(* CoDeSys 2.3.9.41 project: FirstProg.pro *)
(* Libraries: STANDARD.LIB 5.6.98 12:03:02 *)

(* Task configuration *)
TASK Standard (PRIORITY := 0, INTERVAL := T#5ms);
	MAIN
END_TASK

(* Global variable list: Globale_Variablen *)
	VAR_GLOBAL
	globButtonYellow AT %I* : BOOL;
	globButtonBlue AT %I* : BOOL ;
	globLightGreen AT %Q* : BOOL;
	globLightRed AT %Q*  : BOOL;
	globAnalogOutput AT%Q* : INT;
END_VAR

VAR_GLOBAL
	analogOutputMaxVolt : INT :=10 ;
	intMaxValue : INT := 16#7FFF;
	samplingTime : REAL :=0.005;
END_VAR

(* Global variable list: TwinCAT_Configuration *)
(* Generated automatically by TwinCAT - (read only) *)
VAR_CONFIG
	.globButtonYellow AT %IX0.0 : BOOL;	(*  ~ {LinkedWith:TIID^Device 1 (EtherCAT)^Term 1 (EK1200)^Term 2 (EL1004)^Channel 1^Input} *)
	.globButtonBlue AT %IX0.1 : BOOL;	(*  ~ {LinkedWith:TIID^Device 1 (EtherCAT)^Term 1 (EK1200)^Term 2 (EL1004)^Channel 2^Input} *)
	.globLightGreen AT %QX0.0 : BOOL;	(*  ~ {LinkedWith:TIID^Device 1 (EtherCAT)^Term 1 (EK1200)^Term 3 (EL2004)^Channel 1^Output} *)
	.globLightRed AT %QX0.1 : BOOL;	(*  ~ {LinkedWith:TIID^Device 1 (EtherCAT)^Term 1 (EK1200)^Term 3 (EL2004)^Channel 2^Output} *)
	.globAnalogOutput AT %QB4 : INT;	(*  ~ {LinkedWith:TIID^Device 1 (EtherCAT)^Term 1 (EK1200)^Term 5 (EL4034)^AO Outputs Channel 1^Analog output} *)
END_VAR

(* POU MAIN, ST *)
PROGRAM MAIN
VAR
	myBlock : addBlock;
	test : REAL;
END_VAR
UnserProgramm();
myBlock(a := 6.0, b := 6.0);
END_PROGRAM

(* POU addBlock, ST *)
FUNCTION_BLOCK addBlock
VAR_INPUT
	a : REAL;
	b : REAL;
END_VAR
VAR_OUTPUT
	addition : REAL;
	subtraction : REAL;
END_VAR
VAR
END_VAR
addition := a+b;
subtraction := a-b;
END_FUNCTION_BLOCK

(* POU UnserProgramm, ST *)
PROGRAM UnserProgramm
VAR
	intButtonYellowCount : INT := 0;
	Volt : INT;
END_VAR
IF globButtonYellow = TRUE THEN
	globLightGreen := TRUE;
	intButtonYellowCount := intButtonYellowCount + 1;
ELSE
	globLightGreen := FALSE;
END_IF

IF globButtonBlue = TRUE THEN
	globLightRed := TRUE;
	intButtonYellowCount := 0;
ELSE
	globLightRed := FALSE;
END_IF

IF globAnalogOutput.15 THEN
intButtonYellowCount := 0;
END_IF

Volt := intButtonYellowCount / 200;
globAnalogOutput := REAL_TO_INT(((INT_TO_REAL(intButtonYellowCount) /200.0)* INT_TO_REAL(intMaxValue)) / INT_TO_REAL(analogOutputMaxVolt));

(*CASE intButtonYellowCount OF
	0..199 :
	globAnalogOutput := 0;
	200..399 :
	globAnalogOutput := 3277;
	400..599 :
	globAnalogOutput := 6553;
	600..799 :
	globAnalogOutput := 9830;
	800..999 :
	globAnalogOutput := 13107;
	1000..1199 :
	globAnalogOutput := 16384;
	1200..1399 :
	globAnalogOutput := 19660;
	1400..1599 :
	globAnalogOutput := 22937;
	1600..1799 :
	globAnalogOutput := 26214;
	1800..1999 :
	globAnalogOutput := 29490;
	 ELSE
	globAnalogOutput := 32767;
END_CASE*)
END_PROGRAM

(* POU Func, ST *)
FUNCTION Func : REAL
VAR_INPUT
	a : REAL;
	b : REAL;
END_VAR
VAR
END_VAR
Func := a+b;
END_FUNCTION
